# EPICS StreamDevice protocol: code/6.4/temperature.proto
# ./tempApp/Db/temperature.proto
Terminator = CR LF;
get_temp {
   out "T?";
   in  "T %f";
   ExtraInput = Ignore;
}
